// SIMATIC S7-200 project (STEP 7-Micro/WIN), CPU 222 REL 02.01

ORGANIZATION_BLOCK 主程序:OB1
TITLE=程序注释 （可如下更改！！！）
// *VD0为Q0.1、Q0.2、Q0.3、Q0.4延时接通时间；200（模拟值）
// *VD4为Q0.1、Q0.2、Q0.3、Q0.4输出延时时间；300（模拟值）
// *VD8为Q0.0、Q0.1、Q0.2、Q0.3、Q0.4最终延时时间；2000（模拟值）
// *VD12为Q0.0延时接通时间。50（模拟值）
// （1、将HMI指定至上述寄存器，即可改变时间，实现不同时差的工艺要求！）
// （2、本程序由I0.0启动，由I0.1停止。）
BEGIN
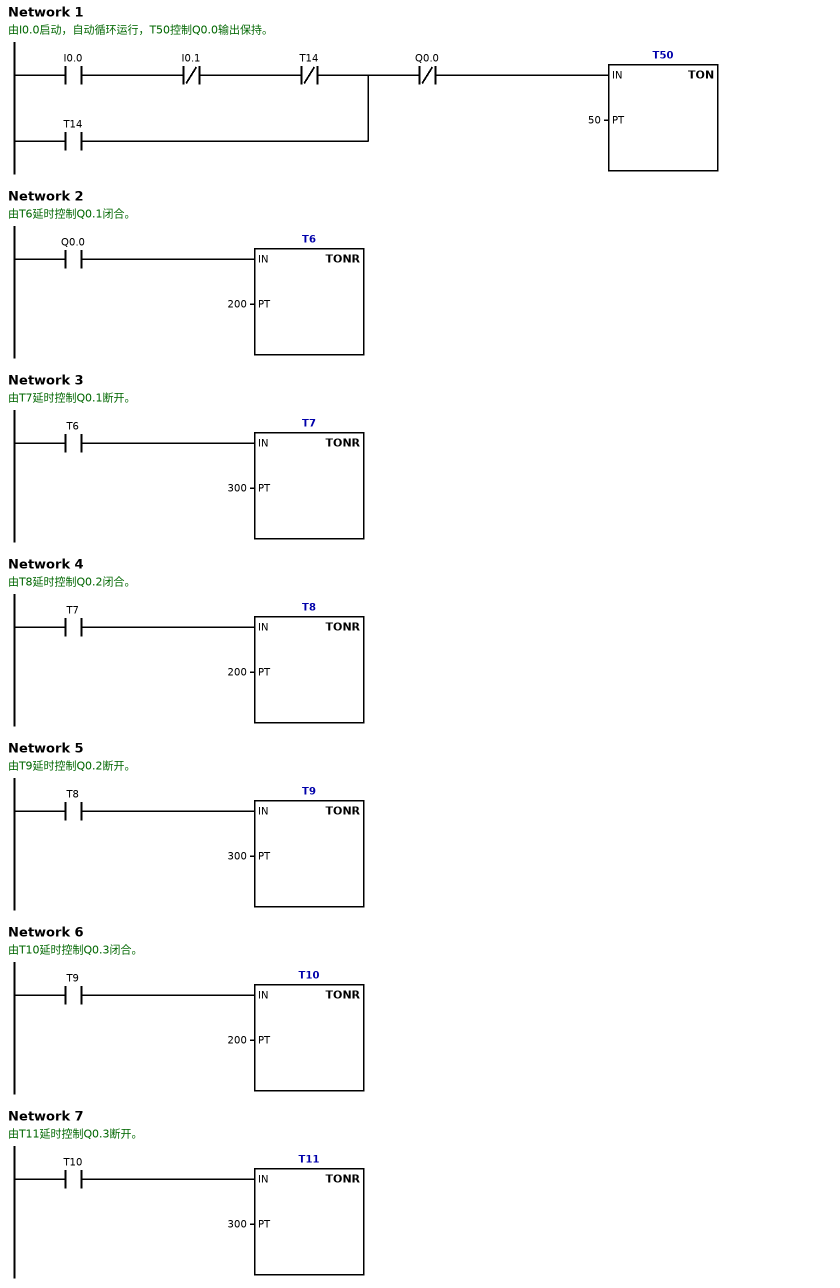
Network 1
// 由I0.0启动，自动循环运行，T50控制Q0.0输出保持。
LD     I0.0
AN     I0.1
AN     T14
O      T14
AN     Q0.0
TON    T50, 50
Network 2
// 由T6延时控制Q0.1闭合。
LD     Q0.0
TONR   T6, 200
Network 3
// 由T7延时控制Q0.1断开。
LD     T6
TONR   T7, 300
Network 4
// 由T8延时控制Q0.2闭合。
LD     T7
TONR   T8, 200
Network 5
// 由T9延时控制Q0.2断开。
LD     T8
TONR   T9, 300
Network 6
// 由T10延时控制Q0.3闭合。
LD     T9
TONR   T10, 200
Network 7
// 由T11延时控制Q0.3断开。
LD     T10
TONR   T11, 300
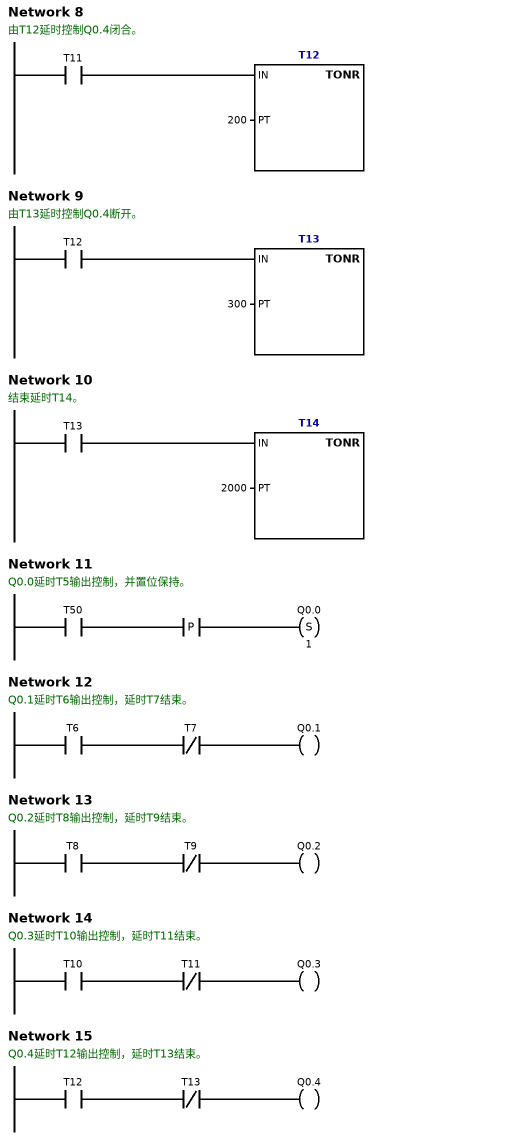
Network 8
// 由T12延时控制Q0.4闭合。
LD     T11
TONR   T12, 200
Network 9
// 由T13延时控制Q0.4断开。
LD     T12
TONR   T13, 300
Network 10
// 结束延时T14。
LD     T13
TONR   T14, 2000
Network 11
// Q0.0延时T5输出控制，并置位保持。
LD     T50
EU
S      Q0.0, 1
Network 12
// Q0.1延时T6输出控制，延时T7结束。
LD     T6
AN     T7
=      Q0.1
Network 13
// Q0.2延时T8输出控制，延时T9结束。
LD     T8
AN     T9
=      Q0.2
Network 14
// Q0.3延时T10输出控制，延时T11结束。
LD     T10
AN     T11
=      Q0.3
Network 15
// Q0.4延时T12输出控制，延时T13结束。
LD     T12
AN     T13
=      Q0.4
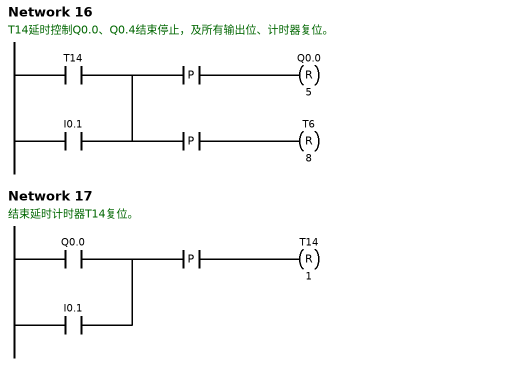
Network 16
// T14延时控制Q0.0、Q0.4结束停止，及所有输出位、计时器复位。
LD     T14
O      I0.1
LPS
EU
R      Q0.0, 5
LPP
EU
R      T6, 8
Network 17
// 结束延时计时器T14复位。
LD     Q0.0
O      I0.1
EU
R      T14, 1
END_ORGANIZATION_BLOCK
